{attribute 'linkalways'} 
{attribute 'no_explicit_call' := 'This FB is a CLASS and must be accessed using methods or properties'}
{attribute 'enable_dynamic_creation'}
FUNCTION_BLOCK _BYTE EXTENDS NumericDatatypeBase
VAR
	localData : BYTE;
	activeData : REFERENCE TO BYTE REF= localData;
END_VAR

PROPERTY PUBLIC Address : PVOID
GET
Address := ADR(activeData);
END_GET
END_PROPERTY

METHOD PUBLIC ClearReference
VAR_INPUT
END_VAR
activeData REF= localData;
END_METHOD

METHOD PUBLIC Clone : I_Datatype
VAR
    pClone : POINTER TO _BYTE;
END_VAR
pClone := __NEW(_BYTE(InitialValue := Value));
Clone := pClone^;
END_METHOD

METHOD FB_init : BOOL
VAR_INPUT
	bInitRetains : BOOL; // if TRUE, the retain variables are initialized (warm start / cold start)
	bInCopyCode : BOOL;  // if TRUE, the instance afterwards gets moved into the copy code (online change)
	InitialValue : BYTE;
END_VAR
localData := InitialValue;
END_METHOD

PROPERTY PUBLIC IsFloat : BOOL
GET
IsFloat := FALSE;
END_GET
END_PROPERTY

PROPERTY PUBLIC IsSigned : BOOL
GET
IsSigned := FALSE;
END_GET
END_PROPERTY

METHOD PUBLIC MakeReferenceTo
VAR_INPUT
	ReferenceTarget : REFERENCE TO BYTE;
END_VAR
activeData REF= ReferenceTarget;
END_METHOD

PROPERTY PUBLIC MaxValue : BYTE
GET
MaxValue := DatatypeLimits.BYTE_MAX_VALUE;
END_GET
END_PROPERTY

PROPERTY PUBLIC MinValue : BYTE
GET
MinValue := DatatypeLimits.BYTE_MIN_VALUE;
END_GET
END_PROPERTY

METHOD PROTECTED SerializeMaxValue
VAR_INPUT
	Serializer : I_Serializer;
END_VAR
Serializer.AddByte(MaxValue);
END_METHOD

METHOD PROTECTED SerializeMinValue
VAR_INPUT
	Serializer : I_Serializer;
END_VAR
Serializer.AddByte(MinValue);
END_METHOD

METHOD PUBLIC SerializeWith
VAR_INPUT
	Serializer : I_Serializer;
END_VAR
Serializer.AddByte(activeData);
END_METHOD

PROPERTY PUBLIC Size : UDINT
GET
Size := SIZEOF(activeData);
END_GET
END_PROPERTY

METHOD TryDeserializeFrom : BOOL
VAR_INPUT
	Deserializer : I_Deserializer;
	Feedback : I_DeserializerFeedback;
END_VAR
TryDeserializeFrom := Deserializer.TryGetByte(activeData, Feedback);
END_METHOD

METHOD TryMakeReferenceTo : BOOL
VAR_INPUT
	Target : I_Datatype;
END_VAR
VAR
	pTargetData : POINTER TO BYTE;
END_VAR
IF NOT (Target.TypeName = TypeName) THEN
	RETURN;
END_IF

pTargetData := Target.Address;
activeData REF= pTargetData^;
TryMakeReferenceTo := TRUE;
END_METHOD

PROPERTY PUBLIC TypeName : T_MAXSTRING
GET
TypeName := 'BYTE';
END_GET
END_PROPERTY

PROPERTY PUBLIC Value : BYTE
GET
Value := activeData;
END_GET
SET
activeData := Value;
END_SET
END_PROPERTY

END_FUNCTION_BLOCK

(* stored: Version 1.1.0.1, ProductVersion 3.1.4024.12
   POU _BYTE: Id {435c7910-bcfd-0b61-1424-a68da74798a8}, SpecialFunc None
   Folder Constructor: Id {10a1f2e3-2a9e-0f3f-1c14-ad6f2f9f2469}
   Folder Protected: Id {c8aa92ee-9999-05e3-3d94-933a58722051}
   Property Address: Id {b66614a5-c3ff-0643-3c72-5cbc61bba641}
   Get Get: Id {95507a03-cf9c-0558-2661-8a3ad4f20f4e}
   Method ClearReference: Id {7a574405-3b90-0edd-1d76-440ed6eff9f1}
   Method Clone: Id {a01b6ab8-1ce2-0028-2130-9f26d5cbeeb1}
   Method FB_init: Id {853cd773-56a1-0625-3b2f-34e410dfc0aa}
   Property IsFloat: Id {27b192cd-5c54-0da5-313f-c38db1571479}
   Get Get: Id {aac9e559-a047-0419-1605-38d0362bf6d9}
   Property IsSigned: Id {c1a0275a-942d-0c9d-1a77-a5ca9d101365}
   Get Get: Id {946a9b2b-557a-08ca-1aad-df9d3ca803d4}
   Method MakeReferenceTo: Id {5aefd03a-0fff-0f66-211c-d5e2c4bb68cb}
   Property MaxValue: Id {05dd455b-32d2-0788-2d0d-89d2aa4a3511}
   Get Get: Id {fc94c668-48e5-0e98-32ac-8b89f4120daf}
   Property MinValue: Id {f2a63b20-1f5c-0c7a-2c87-2d6d4ad85dcd}
   Get Get: Id {c9360b68-0054-0210-2355-fe378193bacf}
   Method SerializeMaxValue: Id {692e460f-5f1f-023f-2111-d3903c907ce8}
   Method SerializeMinValue: Id {29d35e7f-ffb1-029f-1ba1-a688753b6f5d}
   Method SerializeWith: Id {24f8821d-1f88-0d56-1993-dbf051c1d566}
   Property Size: Id {3d96afee-eb4d-07ce-08fb-ff5ea4850ef1}
   Get Get: Id {508eb7ce-422f-0164-1c0d-27697a21df7b}
   Method TryDeserializeFrom: Id {af66ddf6-f930-04e9-3e35-091c1c33f084}
   Method TryMakeReferenceTo: Id {9e7fb14e-b46e-0680-00a7-a8f560d1130f}
   Property TypeName: Id {5e1fb4b4-8820-090a-3c05-c86644a4c87e}
   Get Get: Id {6d3956ea-5b00-0900-2472-25cbe057e6b2}
   Property Value: Id {6c17dd22-4cad-007d-0046-70321a966ab5}
   Get Get: Id {0181aa03-cc31-05a8-22e3-8f7d9332422c}
   Set Set: Id {701a2989-ab2a-0a99-0765-a6eb06d2feee} *)
